PROGRAM MAIN
VAR



// DL Servo
	
{attribute 'OPC.UA.DA':='1'}

DL_Servo_1: FB_MOTOR;

// DL Newport stepper
	
{attribute 'OPC.UA.DA':='1'}
DL_2: FB_MOTOR;

// Camera triggers

//bCameraIN_1 AT %I* : BOOL;

//bCameraIN_2 AT %I* : BOOL;

//bCameraOUT_1 AT %Q* : BOOL;

//bCameraOUT_2 AT %Q* : BOOL;

//{attribute 'OPC.UA.DA':='1'}
//b_Camera_in_1 :BOOL;
//{attribute 'OPC.UA.DA':='1'}
//b_Camera_in_2 :BOOL;
//{attribute 'OPC.UA.DA':='1'}
//b_Camera_out_1 :BOOL;
//{attribute 'OPC.UA.DA':='1'}
//b_Camera_out_2 :BOOL;

{attribute 'OPC.UA.DA':='1'}
fbCryoState : FB_Cryostat_State;

// Homming
iLocalCOntrolStatus : INT;


//Fring Scanning

// Time Stamp
fbGetSystemTime  : GETSYSTEMTIME;
fileTime         : T_FILETIME;
{attribute 'OPC.UA.DA':='1'}
sTime            : STRING;

// NPT PTP

time_info:	FB_TIME;

///

// Filter Wheel

FILTER_WHEEL	:	FB_SCIFY_FILTER_WHEEL_FW102C;

// Accelerometer

in_nVib_X AT %I* :DINT;	
in_nVib_Y AT %I* :DINT;
in_nVib_Z AT %I* :DINT;

{attribute 'OPC.UA.DA':='1'}
nVib_X:	DINT;
{attribute 'OPC.UA.DA':='1'}
nVib_Y:	DINT;
{attribute 'OPC.UA.DA':='1'}
nVib_Z:	DINT;

////
//Shutters
//////
{attribute 'OPC.UA.DA':='1'}
shutter_1:		FB_SHUTTER;


/// Tip-tilt motors
{attribute 'OPC.UA.DA':='1'}
tiptilt_1: FB_MOTOR;




END_VAR


fbCryoState();

DL_Servo_1(sName:='DL_Servo_1', nNOVRAM_DevId:=5, nNOVRAM_Offset:= 1000);

DL_2(sName:='DL_2_Newport', nNOVRAM_DevId:=5, nNOVRAM_Offset:= 2000);

//bCameraOUT_1 := GVL_DL_Scanning_Homming.bTrigCameraImages;


// Time Stamps

fbGetSystemTime(timeLoDW=>fileTime.dwLowDateTime, timeHiDW=>fileTime.dwHighDateTime );
sTime := SYSTEMTIME_TO_STRING( FILETIME_TO_SYSTEMTIME( fileTime ) );

time_info();

// Filter Wheel

FILTER_WHEEL(in_bSimulation:= FALSE, in_sName:= 'FILTER_WHEEL', in_nPeriod:= 1200);

// Vibration from Accelero sensor

nVib_X := in_nVib_X;
nVib_Y := in_nVib_Y;
nVib_Z := in_nVib_Z;

////  Shutters

shutter_1(
	in_sName:= 'Shutter_1', 
	in_bActiveLowClosed:= , 
	in_bActiveLowFault:= , 
	in_bActiveLowOpen:= TRUE, 
	in_bActiveLowSwitch:= , 
	in_bIgnoreClosed:= , 
	in_bIgnoreFault:= , 
	in_bIgnoreOpen:= , 
	in_bInitialState:= , 
	in_nTimeout:= , 
	in_bLogExtTime:= , 
	in_bLog:= );
	
/// Tip-tilt motors

tiptilt_1(sName:='Tip-Tilt_1', nNOVRAM_DevId:=5, nNOVRAM_Offset:= 4000);


//b_Camera_in_1 :=   bCameraIN_1; 

//b_Camera_in_2 :=   bCameraIN_2; 

//b_Camera_out_1 :=  bCameraOUT_1;

//b_Camera_out_2 :=  bCameraOUT_2;

END_PROGRAM

(* stored: Version 1.1.0.1, ProductVersion 3.1.4024.12
   POU MAIN: Id {8b2c4933-f457-4550-be30-efaabcef5e69}, SpecialFunc None *)
